(* PLC project ConveyorCellPLCopen, OpenPLC OpenPLC Editor 1.0 *)
(* stored: creationDateTime 2026-06-17T08:00:00 *)

PROGRAM ConveyorControl
  VAR
    StartPB : BOOL;  (* operator start pushbutton *)
    EStopOK : BOOL;  (* emergency-stop circuit healthy *)
    AutoMode : BOOL;
    JamPhotoeye : BOOL;
    MotorRun : BOOL;  (* conveyor VFD run command *)
    ConvFault : BOOL;
    VFD_Frequency : REAL;  (* drive output frequency Hz *)
    VFD_Current : REAL;
    VFD_FaultCode : DINT;  (* active drive fault code *)
  END_VAR
  VAR_GLOBAL
    LineSpeedSetpoint : REAL := 60.0;
  END_VAR

            IF StartPB AND EStopOK AND AutoMode AND NOT ConvFault THEN
    MotorRun := TRUE;
END_IF;
IF VFD_FaultCode > 0 OR (MotorRun AND JamPhotoeye) THEN
    ConvFault := TRUE;
END_IF;
          
END_PROGRAM
